{attribute 'qualified_only'}
VAR_GLOBAL
	stAxis1: AXIS_REF;
	bButtonFw AT %I*: BOOL; //Self reset
	bButtonBw AT %I*: BOOL; //Self reset
	bButtonHalt AT %I*: BOOL; //Self reset
	bButtonAuto AT %I*: BOOL; //Latch
END_VAR

(* stored: Version 1.1.0.1, ProductVersion 3.1.4024.12
   GVL GVL_MotorDrive: Id {b4228d9d-a8d1-4c04-9422-962d8818e911} *)
